(* CoDeSys 2.3 library: TcMouseEvents.lib *)
(* Libraries: STANDARD.LIB 5.6.98 12:03:02 *)

(* Data type *)
TYPE MouseEvent :
STRUCT
	dwCounter : DWORD; (* The number of events since startup *)
	nXPos : INT; (* The x position of the event *)
	nYPos : INT; (* The y position of the event *)
END_STRUCT
END_TYPE

(* POU MAIN, ST *)
PROGRAM MAIN
VAR
END_VAR
;
END_PROGRAM

(* POU GetLastLeftMouseDownEvent, ST *)
FUNCTION GetLastLeftMouseDownEvent : BOOL
VAR_INPUT
	pMouseEvent : POINTER TO MOUSEEVENT;
END_VAR
VAR
END_VAR
;
END_FUNCTION

(* POU GetLastLeftMouseUpEvent, ST *)
FUNCTION GetLastLeftMouseUpEvent : BOOL
VAR_INPUT
	pMouseEvent : POINTER TO MOUSEEVENT;
END_VAR
VAR
END_VAR
;
END_FUNCTION

(* POU GetLastMouseMoveEvent, ST *)
FUNCTION GetLastMouseMoveEvent : BOOL
VAR_INPUT
	pMouseEvent : POINTER TO MOUSEEVENT;
END_VAR
VAR
END_VAR
;
END_FUNCTION

(* POU GetLastRightMouseDownEvent, ST *)
FUNCTION GetLastRightMouseDownEvent : BOOL
VAR_INPUT
	pMouseEvent : POINTER TO MOUSEEVENT;
END_VAR
VAR
END_VAR
;
END_FUNCTION

(* POU GetLastRightMouseUpEvent, ST *)
FUNCTION GetLastRightMouseUpEvent : BOOL
VAR_INPUT
	pMouseEvent : POINTER TO MOUSEEVENT;
END_VAR
VAR
END_VAR
;
END_FUNCTION

(* POU MouseShowCursor, ST *)
FUNCTION MouseShowCursor : BOOL
VAR_INPUT
	bShow : BOOL;
END_VAR
VAR
END_VAR
;
END_FUNCTION

(* POU SetWindowToForeground, ST *)
FUNCTION SetWindowToForeground : BOOL
VAR_INPUT
	byDummy : BYTE;
END_VAR
VAR
END_VAR
;
END_FUNCTION

(* POU UseSIP, ST *)
FUNCTION UseSIP : BOOL
VAR_INPUT
	byDummy : BYTE;
END_VAR
VAR
END_VAR
;
END_FUNCTION
